Fanuc KAREL source: KA00039.KL

PROGRAM KA00039
%NOLOCKGROUP
VAR
  SRC: STRING[80]
  DST: BOOLEAN
BEGIN
  SRC = 'A'
  DST = SRC
END KA00039
